// Mitsubishi GX Works2 project: nand_2inputs   PLC: Q03UDV
// LRI_2023

PROGRAM MAIN
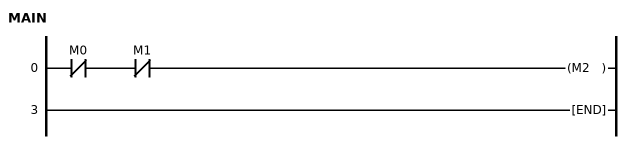
0     LDI     M0
      ANI     M1
      OUT     M2
3     END
END_PROGRAM
